FUNCTION_BLOCK FB_PLCopenCommand_Test EXTENDS TcUnit.FB_TestSuite
VAR_INPUT
END_VAR
VAR_OUTPUT
END_VAR
VAR
END_VAR

// Copyright (c) 2024 Loupe (https://loupe.team), provided under the MIT License.

CallFinished();
CallAbort();
CallError();
AbortPrevious();

METHOD AbortPrevious
VAR
    command : PLCopenCommand();
    newCommand : PLCopenCommand();
END_VAR
// Copyright (c) 2024 Loupe (https://loupe.team), provided under the MIT License.

(*STweep.Disable*)

TEST('AbortPrevious');
	command.Execute := TRUE;
	command();
	command.AbortPreviousCommands(newCommand);
	AssertEquals_DINT(Expected := PLCopenStatusBase.ABORTED, Actual := command.status, Message := 'Initial command should be aborted');
TEST_FINISHED();
END_METHOD

METHOD CallAbort
VAR
    command : PLCopenCommand();
END_VAR
// Copyright (c) 2024 Loupe (https://loupe.team), provided under the MIT License.

(*STweep.Disable*)

TEST('CallAbort');
	AssertFalse(Condition := command.Consume, Message := 'Consume Should start false');
	AssertEquals_DINT(Actual := command.status, Expected:= PLCopenStatusBase.NOT_ENABLED, Message := 'Status should be not enabled');
	
	command.Execute := TRUE;
	
	AssertEquals_DINT(Actual := command.status, Expected:= PLCopenStatusBase.ENABLED_WAITING, Message := 'Status should be waiting');
	
	AssertTrue(Condition := command.Consume, Message := 'Consume Should start as true');
	AssertEquals_DINT(Actual := command.status, Expected:= PLCopenStatusBase.BUSY, Message := 'Status should be busy');
	
	AssertFalse(Condition := command.Consume, Message := 'Consume Should auto reset');
	AssertEquals_DINT(Actual := command.status, Expected:= PLCopenStatusBase.BUSY, Message := 'Status should be busy');
	
	command.Execute := TRUE;
	
	AssertEquals_DINT(Actual := command.status, Expected:= PLCopenStatusBase.ENABLED_WAITING, Message := 'Status should be waiting');
	
	AssertTrue(Condition := command.Consume, Message := 'Consume Should start as true after abort');
	AssertEquals_DINT(Actual := command.status, Expected:= PLCopenStatusBase.BUSY, Message := 'Status should be busy');
	
	AssertFalse(Condition := command.Consume, Message := 'Consume Should auto reset');
	AssertEquals_DINT(Actual := command.status, Expected:= PLCopenStatusBase.BUSY, Message := 'Status should be busy');
	
	command.Finished();
	
	AssertEquals_DINT(Actual := command.status, Expected:= PLCopenStatusBase.ERR_OK, Message := 'Status should be OK after finish');
	command();
	AssertEquals_DINT(Actual := command.status, Expected:= PLCopenStatusBase.NOT_ENABLED, Message := 'Status should auto reset');
	
	AssertFalse(Condition := command.Consume, Message := 'Consume Should auto reset');
	
TEST_FINISHED();
END_METHOD

METHOD CallError
VAR
    command : PLCopenCommand();
END_VAR
// Copyright (c) 2024 Loupe (https://loupe.team), provided under the MIT License.

(*STweep.Disable*)

TEST('CallError');

	AssertFalse(Condition := command.Consume, Message := 'Consume Should start false');
	AssertEquals_DINT(Actual := command.status, Expected:= PLCopenStatusBase.NOT_ENABLED, Message := 'Status should be not enabled');
	
	command.Execute := TRUE;
	
	AssertEquals_DINT(Actual := command.status, Expected:= PLCopenStatusBase.ENABLED_WAITING, Message := 'Status should be waiting');
	
	AssertTrue(Condition := command.Consume, Message := 'Consume Should start as true');
	AssertEquals_DINT(Actual := command.status, Expected:= PLCopenStatusBase.BUSY, Message := 'Status should be busy');
	
	AssertFalse(Condition := command.Consume, Message := 'Consume Should auto reset');
	AssertEquals_DINT(Actual := command.status, Expected:= PLCopenStatusBase.BUSY, Message := 'Status should be busy');
	
	command.Errored(PLCopenStatusBase.ERROR);
	
	AssertFalse(Condition := command.Consume, Message := 'Consume Should be false');
	AssertEquals_DINT(Actual := command.status, Expected:= PLCopenStatusBase.ERROR, Message := 'Status should be error');
	command();
	AssertEquals_DINT(Actual := command.status, Expected:= PLCopenStatusBase.NOT_ENABLED, Message := 'Status should auto reset');
	
	command.Finished();
	
	AssertEquals_DINT(Actual := command.status, Expected:= PLCopenStatusBase.NOT_ENABLED, Message := 'Status should be not enabled if it happens after error');
	
	AssertFalse(Condition := command.Consume, Message := 'Consume Should auto reset');

TEST_FINISHED();
END_METHOD

METHOD CallFinished
VAR
    command : PLCopenCommand();
END_VAR
// Copyright (c) 2024 Loupe (https://loupe.team), provided under the MIT License.

(*STweep.Disable*)

TEST('CallFinished');
	AssertFalse(Condition := command.Consume, Message := 'Consume should start false');
	AssertEquals_DINT(Actual := command.status, Expected:= PLCopenStatusBase.NOT_ENABLED, Message := 'Status should be not enabled');
	
	command.Execute := TRUE;
	
	AssertEquals_DINT(Actual := command.status, Expected:= PLCopenStatusBase.ENABLED_WAITING, Message := 'Status should be waiting');
	
	AssertTrue(Condition := command.Consume, Message := 'Consume should start as true');
	AssertEquals_DINT(Actual := command.status, Expected:= PLCopenStatusBase.BUSY, Message := 'Status should be busy');
	
	AssertFalse(Condition := command.Consume, Message := 'Consume should auto reset');
	AssertEquals_DINT(Actual := command.status, Expected:= PLCopenStatusBase.BUSY, Message := 'Status should be busy');
	
	command.Finished();
	AssertEquals_DINT(Actual := command.status, Expected:= PLCopenStatusBase.ERR_OK, Message := 'Status should be OK after finish');
	command();
	AssertEquals_DINT(Actual := command.status, Expected:= PLCopenStatusBase.NOT_ENABLED, Message := 'Status should auto reset');
	
	AssertFalse(Condition := command.Consume, Message := 'Consume should auto reset');

TEST_FINISHED();
END_METHOD

END_FUNCTION_BLOCK

(* stored: Version 1.1.0.1
   POU FB_PLCopenCommand_Test: Id {0f0750ea-d1ee-4a18-8aa2-27762e9d8df2}, SpecialFunc None
   Method AbortPrevious: Id {5caf9c09-4d16-4f97-b4a8-afa5a2f2097d}
   Method CallAbort: Id {411b9336-d620-4448-b02d-c7622c01b45e}
   Method CallError: Id {1a56507b-64b6-4d10-a688-45cc5b0dc888}
   Method CallFinished: Id {25b22591-3533-478f-bf71-aa6877370f35} *)
